{attribute 'Tc2GvlVarNames'}
VAR_GLOBAL CONSTANT
	(* WT_Zustand_Status *)
	E_WT_Zustand_Status_Idle_Sperre				: SINT := 0;
	E_WT_Zustand_Status_Betriebsbereit			: SINT := 1;
	E_WT_Zustand_Status_Nachl					: SINT := 2;
	E_WT_Zustand_Status_Vorl					: SINT := 3;
	E_WT_Zustand_Status_Betrieb					: SINT := 4;
	E_WT_Zustand_Status_Betrieb_Sperre			: SINT := 5;
	E_WT_Zustand_Status_Stoerung				: SINT := 99;

	(* System_WT_Zustand_Status *)
	E_System_WT_Zustand_Status_Idle_Sperre			: SINT := 0;
	E_System_WT_Zustand_Status_Betriebsbereit		: SINT := 1;
	E_System_WT_Zustand_Status_Nachl_Stellventile	: SINT := 2;
	E_System_WT_Zustand_Status_Vorl_Stellventile	: SINT := 3;
	E_System_WT_Zustand_Status_Nachl_Pumpen			: SINT := 4;
	E_System_WT_Zustand_Status_Vorl_Pumpen			: SINT := 5;
	E_System_WT_Zustand_Status_Betrieb				: SINT := 8;
	E_System_WT_Zustand_Status_Betrieb_Sperre		: SINT := 9;
	E_System_WT_Zustand_Status_Stoerung				: SINT := 99;
END_VAR

(* stored: Version 1.1.0.1, ProductVersion 3.1.4024.9
   GVL Con_WT: Id {e1f9cbb6-d0ea-4e34-954a-fbfee12f5050} *)
